Omron Sysmac Studio project SPA_P5 (Sysmac Studio 1.23.0.14, StandardProject)

# Controller new_Controller_0: NX1P2-1040DT1 version 1.18
Task PrimaryTask (priority 4, period or condition 2000): Programa0

VAR_GLOBAL
    PM : BOOL;  (* Pulsador de Marcha; at BuiltInIO://cpu/#0/Input_Bit_00 *)
    PP : BOOL;  (* Pulsador de Paro; at BuiltInIO://cpu/#0/Input_Bit_01 *)
    O0 : BOOL;  (* Salida 0; at BuiltInIO://cpu/#0/Output_Bit_00 *)
    O1 : BOOL;  (* Salida 1; at BuiltInIO://cpu/#0/Output_Bit_01 *)
    HMI_PM AT %W0.0 : BOOL;  (* published *)
    HMI_PP AT %W0.1 : BOOL;  (* published *)
    HMI_O0 AT %W1.0 : BOOL;  (* published *)
    HMI_O1 AT %W1.1 : BOOL;  (* published *)
END_VAR
VAR_GLOBAL RETAIN
    HMI_Temperatura AT %D0 : INT;  (* published *)
    HMI_Humedad AT %D2 : INT;  (* published *)
END_VAR

PROGRAM Programa0
VAR
    hmi : BOOL;
    Temperatura : INT;
    Humedad : INT;
END_VAR
VAR_EXTERNAL
    PM : BOOL;
    PP : BOOL;
    O0 : BOOL;
    HMI_PM : BOOL;
    HMI_O0 : BOOL;
    HMI_PP : BOOL;
    HMI_Temperatura : INT;
    HMI_Humedad : INT;
END_VAR
VAR
    _p1 : BOOL;
END_VAR

(* Section Sección0: ladder, written here as Structured Text *)

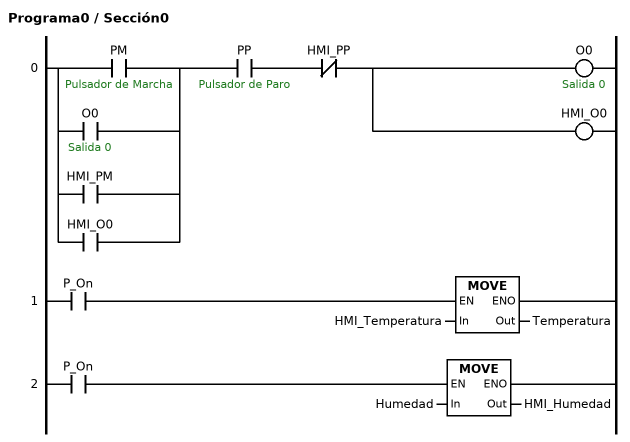
(* Rung 0 *)
_p1 := (PM OR O0 OR HMI_PM OR HMI_O0) AND PP AND NOT HMI_PP;
O0 := _p1;
HMI_O0 := _p1;
(* Rung 1 *)
IF P_On THEN Temperatura := HMI_Temperatura; END_IF;
(* Rung 2 *)
IF P_On THEN HMI_Humedad := Humedad; END_IF;
END_PROGRAM